FUNCTION_BLOCK FB_Refactoring
VAR_INPUT
	i_a  :BOOL;
    i_b  :BOOL;
    i_c  :BOOL;
    i_d  :BOOL;
    i_e  :BOOL;
    i_f  :BOOL;
   
END_VAR
VAR_OUTPUT
	q_a   :BOOL;
    q_b   :BOOL;
    q_c   :BOOL;
END_VAR
VAR
	ref_Dummy	: FB_RefDummy;
END_VAR

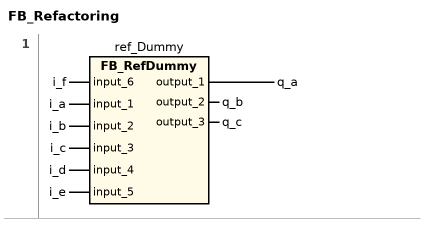
// NETWORK 1
ref_Dummy(
    input_6 := i_f,
    input_1 := i_a,
    input_2 := i_b,
    input_3 := i_c,
    input_4 := i_d,
    input_5 := i_e,
    output_2 => q_b,
    output_3 => q_c); // FB_RefDummy
q_a := ref_Dummy.output_1;

END_FUNCTION_BLOCK

(* stored: Version 1.1.0.1, ProductVersion 3.1.4024.12
   POU FB_Refactoring: Id {9c23e4b1-adf3-4510-bd05-bee0da6456e5}, SpecialFunc None *)
